VAR_GLOBAL
	LogToTextBuffer		: ST_String_FIFO;	// Text log
	fbLocalTime			: FB_LocalSystemTime;
END_VAR

(* stored: Version 1.1.0.1, ProductVersion 3.1.4024.5
   GVL GVL_Log: Id {d2e63ab5-6f42-4229-bf4f-3a9b255a5e88} *)
